Fanuc KAREL source: kt00440.KL

PROGRAM KT00440
%STACKSIZE=65535
%PRIORITY=65535
%NOLOCKGROUP
VAR
I1 : INTEGER
OUT : BOOLEAN
-- UNRESOLVED DECLARATIONS (source type spelling not recovered)
-- H2 : ARRAY[2] OF TYPE_0x0017 (type_u16=0x2017)
BEGIN
I1=2
-- UNRESOLVED_PC line 9 opcodes [2E 22 9D 33 B4] marker_code=16
-- UNRESOLVED_PC line 10 opcodes [21 22 9D 33 B3 5C 23] marker_code=35
END KT00440
